FUNCTION_BLOCK FB_SaMElementProduction EXTENDS FB_SaMElement
VAR
END_VAR

METHOD FB_init : BOOL
VAR_INPUT
	bInitRetains : BOOL; // if TRUE, the retain variables are initialized (warm start / cold start)
	bInCopyCode : BOOL;  // if TRUE, the instance afterwards gets moved into the copy code (online change)
END_VAR
THIS^.SetText (eLocation := E_BaseLocation.pl, wsDescription := "Produkcja");
THIS^.SetText (eLocation := E_BaseLocation.en, wsDescription := "Production");
THIS^.SetText (eLocation := E_BaseLocation.de, wsDescription := "Produktion");
THIS^.SetName (stName := THIS^.GetTexts ());
END_METHOD

END_FUNCTION_BLOCK

(* stored: Version 1.1.0.1
   POU FB_SaMElementProduction: Id {2553c4ee-ccbe-09f4-23d8-9032ffb84f10}, SpecialFunc None
   Method FB_init: Id {669b6434-50b0-0fe6-315d-0e1547e5746f} *)
